// TIA Portal V20 export
DATA_BLOCK "DB_CC_HMI"   // DB100
{ S7_Optimized_Access := 'TRUE' }
// stored: AutoNumber false, MemoryReserve 100
   VAR
      Safety_ACK : Bool;
      Reset_Drives : Bool;
      Reset_Safety : Bool;
      Error_Status : Bool;
      CC_ST23_RollsUp : Bool;
      CC_ST23_RollsDown : Bool;
      CC_ST23_ModulesUp : Bool;
      CC_ST23_ModulesDown : Bool;
      CC_ST23_Wibrating : Bool;
      CC_ST23_DriveRollerUp : Bool;
      CC_ST23_DriveRollerDown : Bool;
      CC_ST23_WibratingAuto : Bool;
      CC_ST23_UnlockPallete : Bool;
      CC_ST24_RollsUp : Bool;
      CC_ST24_RollsDown : Bool;
      CC_ST24_ModulesUp : Bool;
      CC_ST24_ModulesDown : Bool;
      CC_ST24_Wibrating : Bool;
      CC_ST24_DriveRollerUp : Bool;
      CC_ST24_DriveRollerDown : Bool;
      CC_ST24_WibratingAuto : Bool;
      CC_ST24_UnlockPallete : Bool;
      CC_ST25_RollsUp : Bool;
      CC_ST25_RollsDown : Bool;
      CC_ST25_ModulesUp : Bool;
      CC_ST25_ModulesDown : Bool;
      CC_ST25_Wibrating : Bool;
      CC_ST25_DriveRollerUp : Bool;
      CC_ST25_DriveRollerDown : Bool;
      CC_ST25_WibratingAuto : Bool;
      CC_ST25_UnlockPallete : Bool;
   END_VAR
BEGIN
END_DATA_BLOCK
